FUNCTION_BLOCK FB_MotorControl_Test EXTENDS FB_TestSuite
VAR_INPUT
END_VAR
VAR_OUTPUT
END_VAR
VAR
END_VAR

TestWhenSensorIsOff();
TestWhenButton1Off();

METHOD TestWhenButton1Off
VAR_INPUT
END_VAR
VAR
	motorControl : FB_MotorControl;
	result : BOOL;
	expected_result : BOOL := TRUE;
	
END_VAR
TEST('TestWhenButton1Off');

motorControl( Button1 := FALSE, Button2 := TRUE, Sensor := FALSE, Motor => result);


AssertEquals(Expected := expected_result,
             Actual := result,
             Message := 'The output is not correct' );

TEST_FINISHED();
END_METHOD

METHOD TestWhenSensorIsOff
VAR_INPUT
END_VAR
VAR
	motorControl : FB_MotorControl;
	result : BOOL;
	expected_result : BOOL := TRUE;
END_VAR
TEST('TestWhenSensorIsOff');

motorControl( Button1 := TRUE, Button2 := TRUE, Sensor := FALSE, Motor => result);
 
AssertEquals(Expected := expected_result,
             Actual := result,
             Message := 'The output is not correct' );
TEST_FINISHED();
END_METHOD

END_FUNCTION_BLOCK

(* stored: Version 1.1.0.1, ProductVersion 3.1.4024.12
   POU FB_MotorControl_Test: Id {5cd1b32c-e14b-4bf7-a757-fc4cfcd8348d}, SpecialFunc None
   Method TestWhenButton1Off: Id {943300ca-156f-47eb-824f-66d8ca86ce3e}
   Method TestWhenSensorIsOff: Id {6db6ec2f-07f1-4bbb-8a1c-16284cff6942} *)
